// TIA Portal V15.1 export
// export: Created 2020-06-12T07:35:42.9130859Z, ExportSetting None, DisplayName Totally Integrated Automation Portal, DisplayVersion V15.1, DisplayName TIA Portal Openness, DisplayVersion V15.1, DisplayName STEP 7 Professional, DisplayVersion V15.1, DisplayName STEP 7 Safety, DisplayVersion V15.1, DisplayName WinCC Advanced, DisplayVersion V15.1
FUNCTION "CW_MS1" : Void   // FC119, FBD
TITLE = Meltstation #1 cooling control
{ S7_Optimized_Access := 'TRUE' }
// stored: SetENOAutomatically False
   VAR_TEMP
      tContReset : Bool;
      tContDTOn : Bool;
      tMoldIsClosed : Bool;
      tMoldIsOpened : Bool;
      tMoldIsDischarging : Bool;
      tMoldIsPrepared : Bool;
      tBaseIsClosed : Bool;
      tBaseIsOpened : Bool;
      tBaseIsPrepared : Bool;
      tBaseIsDischarging : Bool;
      tLinesToOpen : Bool;
      tLinesToCLose : Bool;
      tToDischarge : Bool;
      tCoolingIsOn : Bool;
      tCoolingOn : Bool;
      tCoolingOff : Bool;
      tCoolingLockOff : Bool;
      tDeltaContOn : Bool;
      tStepError : Bool;
      tReqOn : Bool;
      tReqOff : Bool;
      tReqDisStop : Bool;
      tReqDisStart : Bool;
      tValid : Bool;
      tReqContFlow : Bool;
      tReqContDT : Bool;
      tStage : Int;
      tStepInternal : Int;
      tMoldFlowMax : Real;
      tBaseFlowMax : Real;
      tMoldFlowSet : Real;
      tMoldFlowPhysMax : Real;
      tMoldFlowPhysMin : Real;
      tMoldFlowMin : Real;
      tBaseFlowPhysMax : Real;
      tBaseFlowPhysMin : Real;
      tBaseFlowMin : Real;
      tBaseFlowSet : Real;
      tMoldFlowContIsOn : Bool;
      tBaseFlowContOn : Bool;
      tMoldFlowContIsAuto : Bool;
      tEnAlarms : Bool;
      tCopyParam : Bool;
   END_VAR
BEGIN

REGION Network 1: HMI request treat
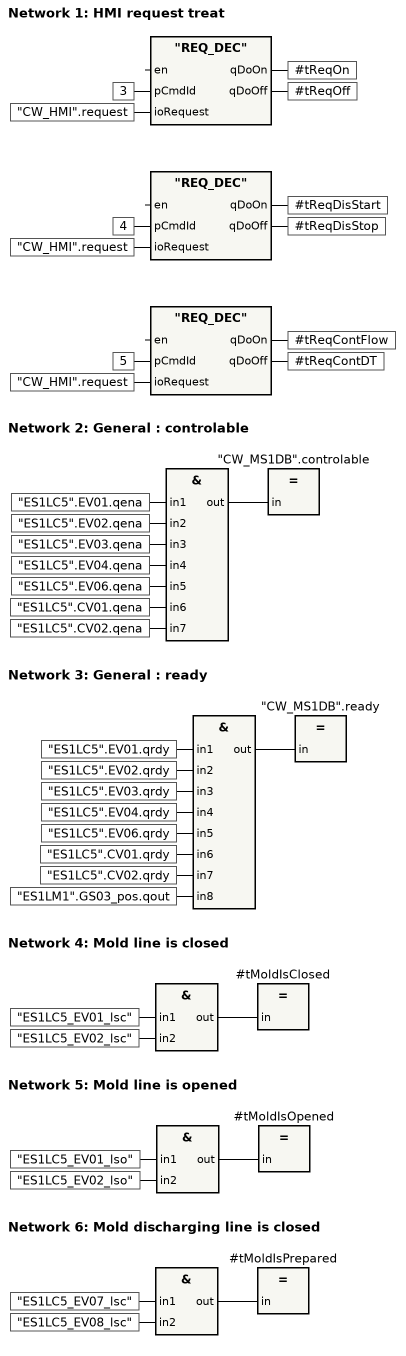
   "REQ_DEC"(pCmdId := 3, ioRequest := "CW_HMI".request, qDoOn => #tReqOn, qDoOff => #tReqOff);
   "REQ_DEC"(pCmdId := 4, ioRequest := "CW_HMI".request, qDoOn => #tReqDisStart, qDoOff => #tReqDisStop);
   "REQ_DEC"(pCmdId := 5, ioRequest := "CW_HMI".request, qDoOn => #tReqContFlow, qDoOff => #tReqContDT);
END_REGION

REGION Network 2: General : controlable
   "CW_MS1DB".controlable := "ES1LC5".EV01.qena AND "ES1LC5".EV02.qena AND "ES1LC5".EV03.qena AND "ES1LC5".EV04.qena AND "ES1LC5".EV06.qena AND "ES1LC5".CV01.qena AND "ES1LC5".CV02.qena;
END_REGION

REGION Network 3: General : ready
   "CW_MS1DB".ready := "ES1LC5".EV01.qrdy AND "ES1LC5".EV02.qrdy AND "ES1LC5".EV03.qrdy AND "ES1LC5".EV04.qrdy AND "ES1LC5".EV06.qrdy AND "ES1LC5".CV01.qrdy AND "ES1LC5".CV02.qrdy AND "ES1LM1".GS03_pos.qout;
END_REGION

REGION Network 4: Mold line is closed
   #tMoldIsClosed := "ES1LC5_EV01_lsc" AND "ES1LC5_EV02_lsc";
END_REGION

REGION Network 5: Mold line is opened
   #tMoldIsOpened := "ES1LC5_EV01_lso" AND "ES1LC5_EV02_lso";
END_REGION

REGION Network 6: Mold discharging line is closed
   #tMoldIsPrepared := "ES1LC5_EV07_lsc" AND "ES1LC5_EV08_lsc";
END_REGION

REGION Network 7: Mold discharging line is opened
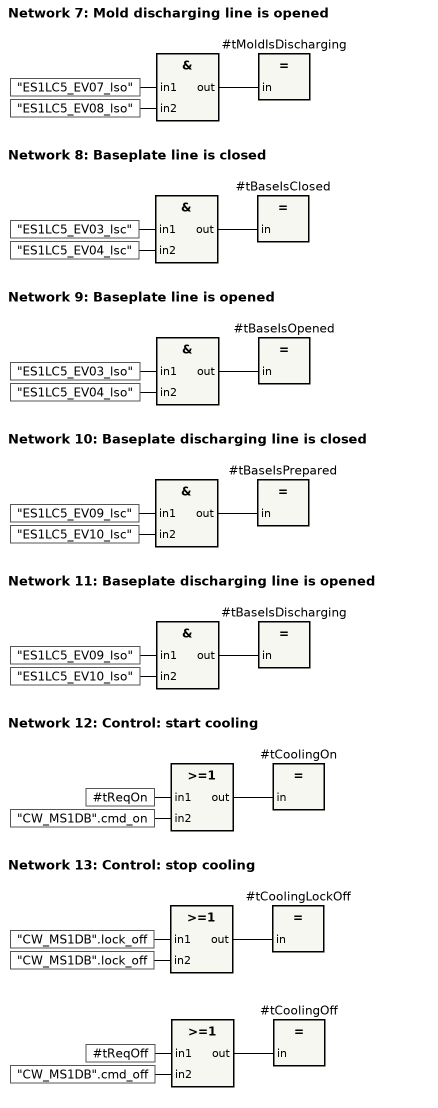
   #tMoldIsDischarging := "ES1LC5_EV07_lso" AND "ES1LC5_EV08_lso";
END_REGION

REGION Network 8: Baseplate line is closed
   #tBaseIsClosed := "ES1LC5_EV03_lsc" AND "ES1LC5_EV04_lsc";
END_REGION

REGION Network 9: Baseplate line is opened
   #tBaseIsOpened := "ES1LC5_EV03_lso" AND "ES1LC5_EV04_lso";
END_REGION

REGION Network 10: Baseplate discharging line is closed
   #tBaseIsPrepared := "ES1LC5_EV09_lsc" AND "ES1LC5_EV10_lsc";
END_REGION

REGION Network 11: Baseplate discharging line is opened
   #tBaseIsDischarging := "ES1LC5_EV09_lso" AND "ES1LC5_EV10_lso";
END_REGION

REGION Network 12: Control: start cooling
   #tCoolingOn := #tReqOn OR "CW_MS1DB".cmd_on;
END_REGION

REGION Network 13: Control: stop cooling
   // #tReqAmcOff
   #tCoolingLockOff := "CW_MS1DB".lock_off OR "CW_MS1DB".lock_off;
   #tCoolingOff := #tReqOff OR "CW_MS1DB".cmd_off;
END_REGION

REGION Network 14: *** Control (stages) ***
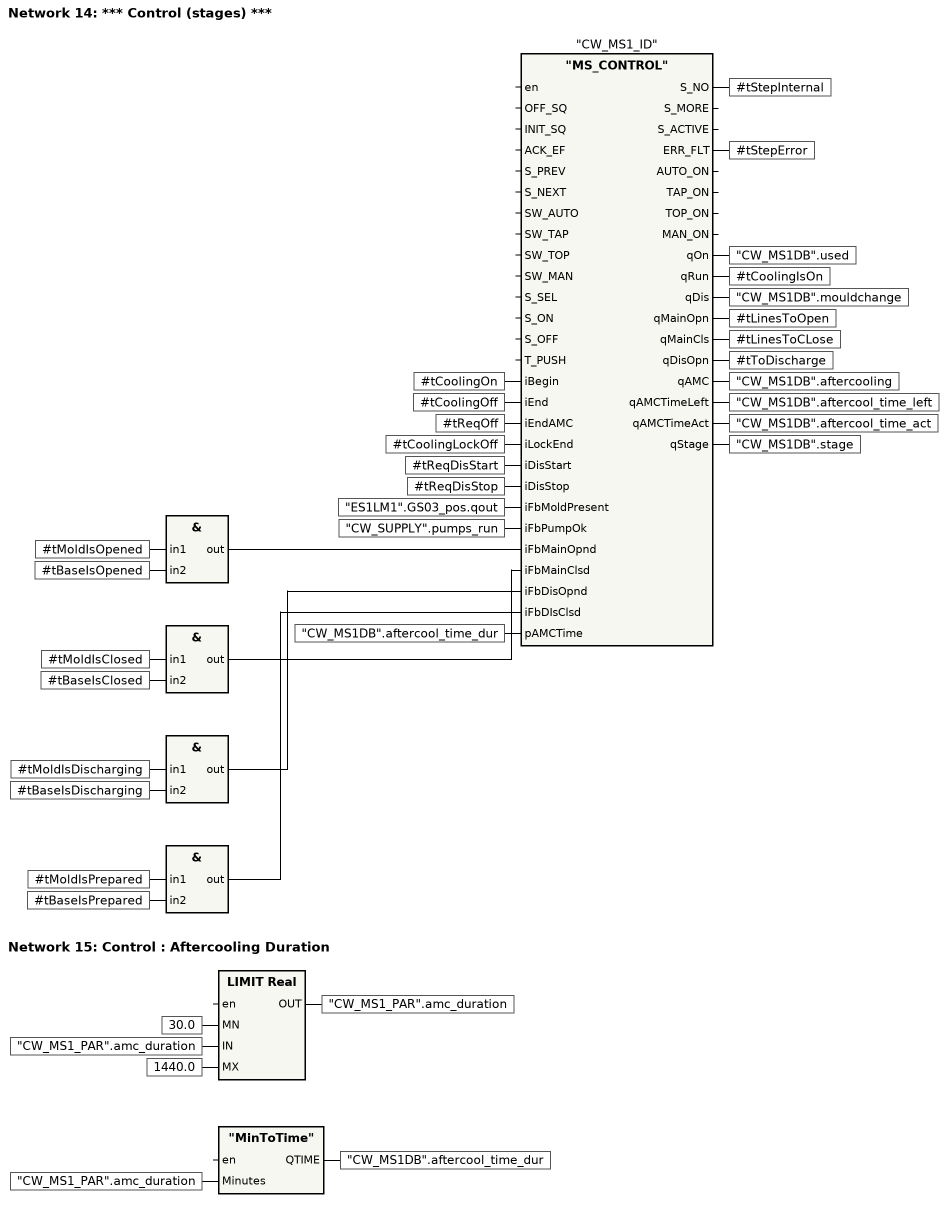
   "CW_MS1_ID"(iBegin := #tCoolingOn,   // "MS_CONTROL"
               iEnd := #tCoolingOff,
               iEndAMC := #tReqOff,
               iLockEnd := #tCoolingLockOff,
               iDisStart := #tReqDisStart,
               iDisStop := #tReqDisStop,
               iFbMoldPresent := "ES1LM1".GS03_pos.qout,
               iFbPumpOk := "CW_SUPPLY".pumps_run,
               iFbMainOpnd := #tMoldIsOpened AND #tBaseIsOpened,
               iFbMainClsd := #tMoldIsClosed AND #tBaseIsClosed,
               iFbDisOpnd := #tMoldIsDischarging AND #tBaseIsDischarging,
               iFbDIsClsd := #tMoldIsPrepared AND #tBaseIsPrepared,
               pAMCTime := "CW_MS1DB".aftercool_time_dur,
               S_NO => #tStepInternal,
               ERR_FLT => #tStepError,
               qOn => "CW_MS1DB".used,
               qRun => #tCoolingIsOn,
               qDis => "CW_MS1DB".mouldchange,
               qMainOpn => #tLinesToOpen,
               qMainCls => #tLinesToCLose,
               qDisOpn => #tToDischarge,
               qAMC => "CW_MS1DB".aftercooling,
               qAMCTimeLeft => "CW_MS1DB".aftercool_time_left,
               qAMCTimeAct => "CW_MS1DB".aftercool_time_act,
               qStage => "CW_MS1DB".stage);
END_REGION

REGION Network 15: Control : Aftercooling Duration
   // Convert minutes to milliseconds
   "CW_MS1_PAR".amc_duration := LIMIT(MN := 30.0, IN := "CW_MS1_PAR".amc_duration, MX := 1440.0);
   "MinToTime"(Minutes := "CW_MS1_PAR".amc_duration, QTIME => "CW_MS1DB".aftercool_time_dur);
END_REGION

REGION Network 16: Cooling mode: flow/delta-T
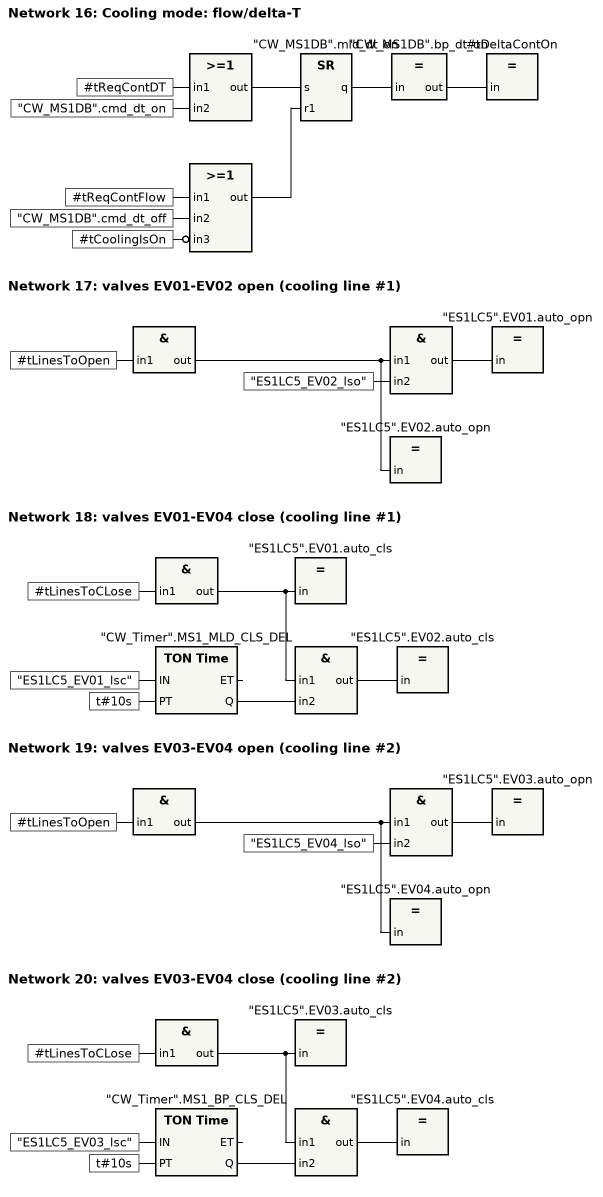
   IF #tReqContDT OR "CW_MS1DB".cmd_dt_on THEN
       "CW_MS1DB".mld_dt_on := TRUE;   // SR flip-flop
   END_IF;
   IF #tReqContFlow OR "CW_MS1DB".cmd_dt_off OR NOT #tCoolingIsOn THEN "CW_MS1DB".mld_dt_on := FALSE; END_IF;
   "CW_MS1DB".bp_dt_on := "CW_MS1DB".mld_dt_on;
   #tDeltaContOn := "CW_MS1DB".mld_dt_on;
END_REGION

REGION Network 17: valves EV01-EV02 open (cooling line #1)
   "ES1LC5".EV01.auto_opn := #tLinesToOpen AND "ES1LC5_EV02_lso";
   "ES1LC5".EV02.auto_opn := #tLinesToOpen;
END_REGION

REGION Network 18: valves EV01-EV04 close (cooling line #1)
   "ES1LC5".EV01.auto_cls := #tLinesToCLose;
   "CW_Timer".MS1_MLD_CLS_DEL.TON(IN := "ES1LC5_EV01_lsc", PT := t#10s);
   "ES1LC5".EV02.auto_cls := #tLinesToCLose AND "CW_Timer".MS1_MLD_CLS_DEL.Q;
END_REGION

REGION Network 19: valves EV03-EV04 open (cooling line #2)
   "ES1LC5".EV03.auto_opn := #tLinesToOpen AND "ES1LC5_EV04_lso";
   "ES1LC5".EV04.auto_opn := #tLinesToOpen;
END_REGION

REGION Network 20: valves EV03-EV04 close (cooling line #2)
   "ES1LC5".EV03.auto_cls := #tLinesToCLose;
   "CW_Timer".MS1_BP_CLS_DEL.TON(IN := "ES1LC5_EV03_lsc", PT := t#10s);
   "ES1LC5".EV04.auto_cls := #tLinesToCLose AND "CW_Timer".MS1_BP_CLS_DEL.Q;
END_REGION

REGION Network 21: valves EV01-EV04 to close lock
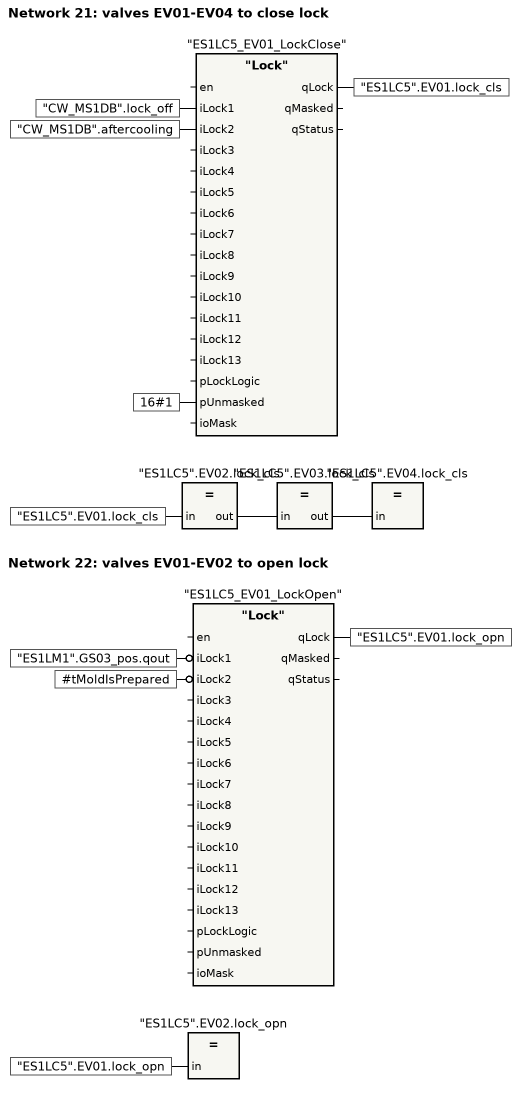
   "ES1LC5_EV01_LockClose"(iLock1 := "CW_MS1DB".lock_off,   // "Lock"
                           iLock2 := "CW_MS1DB".aftercooling,
                           pUnmasked := 16#1,
                           qLock => "ES1LC5".EV01.lock_cls);
   "ES1LC5".EV02.lock_cls := "ES1LC5".EV01.lock_cls;
   "ES1LC5".EV03.lock_cls := "ES1LC5".EV01.lock_cls;
   "ES1LC5".EV04.lock_cls := "ES1LC5".EV01.lock_cls;
END_REGION

REGION Network 22: valves EV01-EV02 to open lock
   "ES1LC5_EV01_LockOpen"(iLock1 := NOT "ES1LM1".GS03_pos.qout,   // "Lock"
                          iLock2 := NOT #tMoldIsPrepared,
                          qLock => "ES1LC5".EV01.lock_opn);
   "ES1LC5".EV02.lock_opn := "ES1LC5".EV01.lock_opn;
END_REGION

REGION Network 23: valves EV03-EV04 to open lock
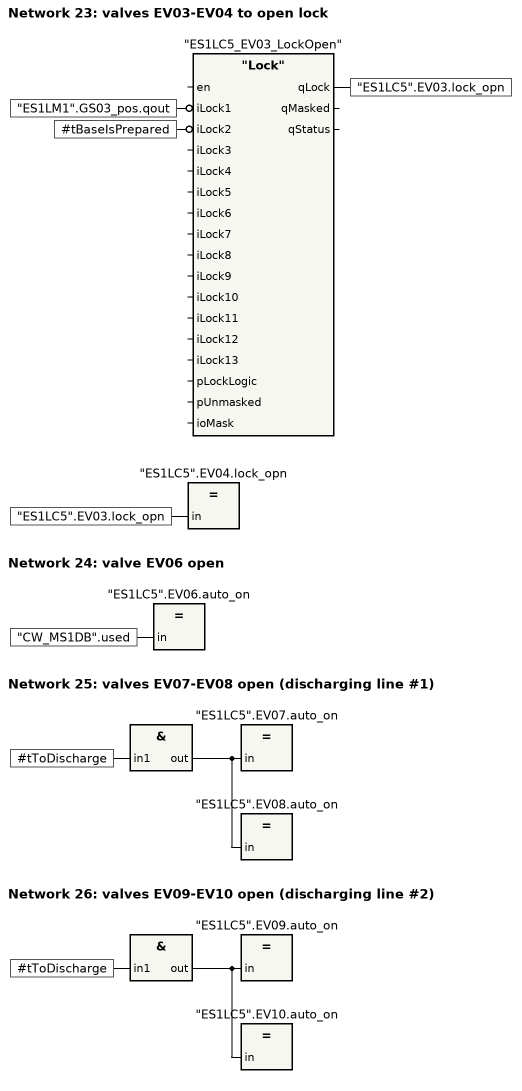
   "ES1LC5_EV03_LockOpen"(iLock1 := NOT "ES1LM1".GS03_pos.qout,   // "Lock"
                          iLock2 := NOT #tBaseIsPrepared,
                          qLock => "ES1LC5".EV03.lock_opn);
   "ES1LC5".EV04.lock_opn := "ES1LC5".EV03.lock_opn;
END_REGION

REGION Network 24: valve EV06 open
   "ES1LC5".EV06.auto_on := "CW_MS1DB".used;
END_REGION

REGION Network 25: valves EV07-EV08 open (discharging line #1)
   "ES1LC5".EV07.auto_on := #tToDischarge;
   "ES1LC5".EV08.auto_on := #tToDischarge;
END_REGION

REGION Network 26: valves EV09-EV10 open (discharging line #2)
   "ES1LC5".EV09.auto_on := #tToDischarge;
   "ES1LC5".EV10.auto_on := #tToDischarge;
END_REGION

REGION Network 27: valves EV07-EV08 to open lock (discharging line #1)
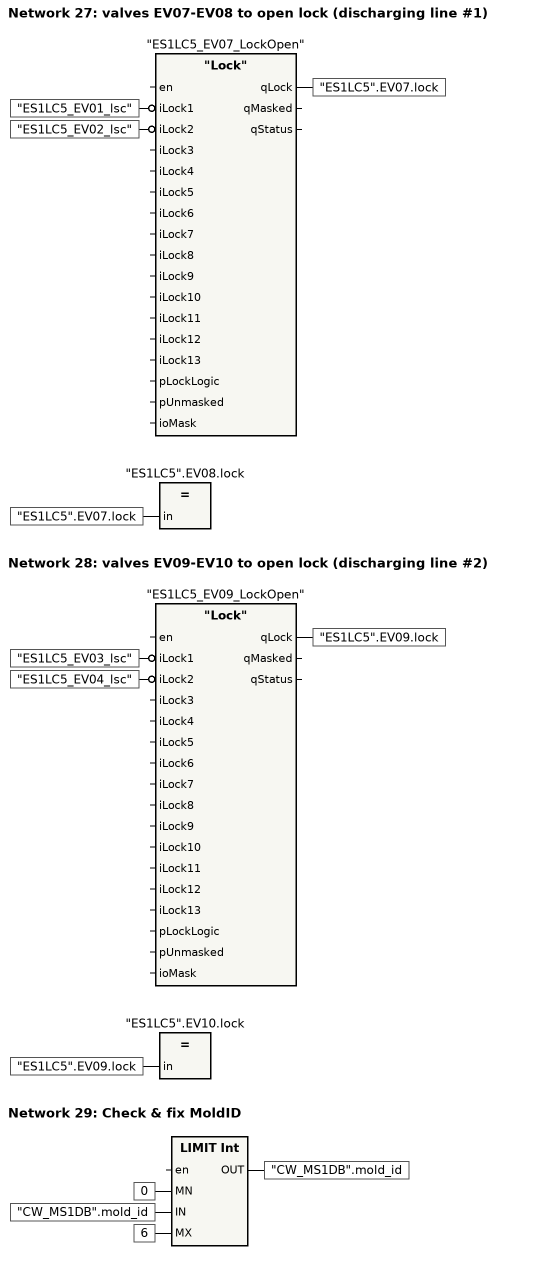
   "ES1LC5_EV07_LockOpen"(iLock1 := NOT "ES1LC5_EV01_lsc",   // "Lock"
                          iLock2 := NOT "ES1LC5_EV02_lsc",
                          qLock => "ES1LC5".EV07.lock);
   "ES1LC5".EV08.lock := "ES1LC5".EV07.lock;
END_REGION

REGION Network 28: valves EV09-EV10 to open lock (discharging line #2)
   "ES1LC5_EV09_LockOpen"(iLock1 := NOT "ES1LC5_EV03_lsc",   // "Lock"
                          iLock2 := NOT "ES1LC5_EV04_lsc",
                          qLock => "ES1LC5".EV09.lock);
   "ES1LC5".EV10.lock := "ES1LC5".EV09.lock;
END_REGION

REGION Network 29: Check & fix MoldID
   "CW_MS1DB".mold_id := LIMIT(MN := 0, IN := "CW_MS1DB".mold_id, MX := 6);
END_REGION

REGION Network 30: MOULD: Setpoint flow mould
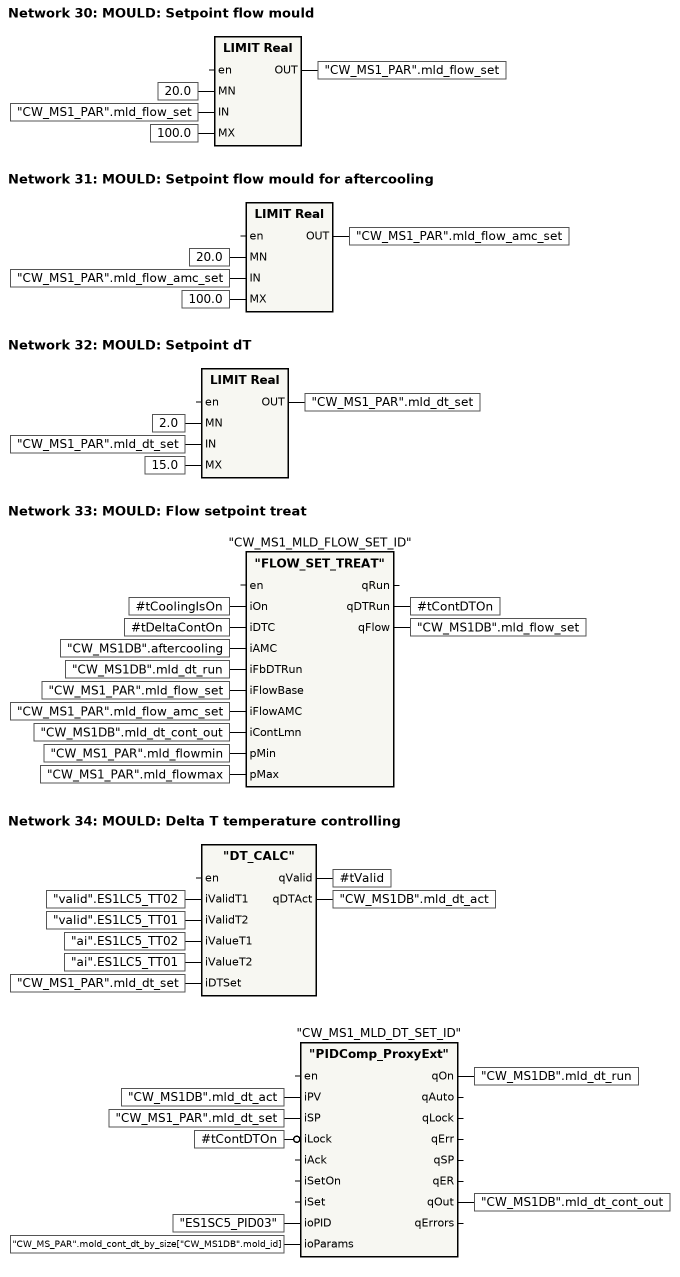
   "CW_MS1_PAR".mld_flow_set := LIMIT(MN := 20.0, IN := "CW_MS1_PAR".mld_flow_set, MX := 100.0);
END_REGION

REGION Network 31: MOULD: Setpoint flow mould for aftercooling
   "CW_MS1_PAR".mld_flow_amc_set := LIMIT(MN := 20.0, IN := "CW_MS1_PAR".mld_flow_amc_set, MX := 100.0);
END_REGION

REGION Network 32: MOULD: Setpoint dT
   "CW_MS1_PAR".mld_dt_set := LIMIT(MN := 2.0, IN := "CW_MS1_PAR".mld_dt_set, MX := 15.0);
END_REGION

REGION Network 33: MOULD: Flow setpoint treat
   "CW_MS1_MLD_FLOW_SET_ID"(iOn := #tCoolingIsOn,   // "FLOW_SET_TREAT"
                           iDTC := #tDeltaContOn,
                           iAMC := "CW_MS1DB".aftercooling,
                           iFbDTRun := "CW_MS1DB".mld_dt_run,
                           iFlowBase := "CW_MS1_PAR".mld_flow_set,
                           iFlowAMC := "CW_MS1_PAR".mld_flow_amc_set,
                           iContLmn := "CW_MS1DB".mld_dt_cont_out,
                           pMin := "CW_MS1_PAR".mld_flowmin,
                           pMax := "CW_MS1_PAR".mld_flowmax,
                           qDTRun => #tContDTOn,
                           qFlow => "CW_MS1DB".mld_flow_set);
END_REGION

REGION Network 34: MOULD: Delta T temperature controlling
   "DT_CALC"(iValidT1 := "valid".ES1LC5_TT02,
             iValidT2 := "valid".ES1LC5_TT01,
             iValueT1 := "ai".ES1LC5_TT02,
             iValueT2 := "ai".ES1LC5_TT01,
             iDTSet := "CW_MS1_PAR".mld_dt_set,
             qValid => #tValid,
             qDTAct => "CW_MS1DB".mld_dt_act);
   "CW_MS1_MLD_DT_SET_ID"(iPV := "CW_MS1DB".mld_dt_act,   // "PIDComp_ProxyExt"
                          iSP := "CW_MS1_PAR".mld_dt_set,
                          iLock := NOT #tContDTOn,
                          ioPID := "ES1SC5_PID03",
                          ioParams := "CW_MS_PAR".mold_cont_dt_by_size["CW_MS1DB".mold_id],
                          qOn => "CW_MS1DB".mld_dt_run,
                          qOut => "CW_MS1DB".mld_dt_cont_out);
END_REGION

REGION Network 35: MOULD: Flow Controller
   // Yes, the actual value is keeping while a measurement is not valid.
   // If the controller is stable (ERR = 0) we can avoid a bump by flow,
   // else if ERR > 0 the controller will open the valve, and this is also not bad
   // else the controller will close the valve, and this is bad...
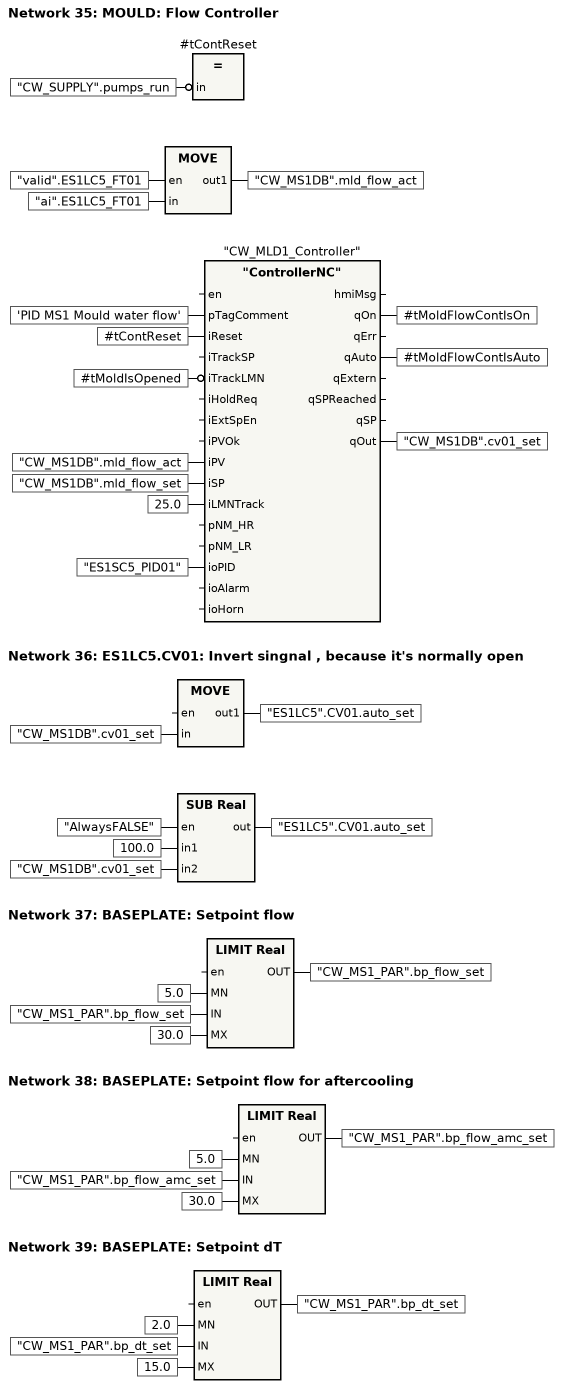
   #tContReset := NOT "CW_SUPPLY".pumps_run;
   IF "valid".ES1LC5_FT01 THEN "CW_MS1DB".mld_flow_act := "ai".ES1LC5_FT01; END_IF;
   "CW_MLD1_Controller"(pTagComment := 'PID MS1 Mould water flow',   // "ControllerNC"
                        iReset := #tContReset,
                        iTrackLMN := NOT #tMoldIsOpened,
                        iPV := "CW_MS1DB".mld_flow_act,
                        iSP := "CW_MS1DB".mld_flow_set,
                        iLMNTrack := 25.0,
                        ioPID := "ES1SC5_PID01",
                        qOn => #tMoldFlowContIsOn,
                        qAuto => #tMoldFlowContIsAuto,
                        qOut => "CW_MS1DB".cv01_set);
END_REGION

REGION Network 36: ES1LC5.CV01: Invert singnal , because it's normally open
   "ES1LC5".CV01.auto_set := "CW_MS1DB".cv01_set;
   IF "AlwaysFALSE" THEN "ES1LC5".CV01.auto_set := 100.0 - "CW_MS1DB".cv01_set; END_IF;
END_REGION

REGION Network 37: BASEPLATE: Setpoint flow
   "CW_MS1_PAR".bp_flow_set := LIMIT(MN := 5.0, IN := "CW_MS1_PAR".bp_flow_set, MX := 30.0);
END_REGION

REGION Network 38: BASEPLATE: Setpoint flow for aftercooling
   "CW_MS1_PAR".bp_flow_amc_set := LIMIT(MN := 5.0, IN := "CW_MS1_PAR".bp_flow_amc_set, MX := 30.0);
END_REGION

REGION Network 39: BASEPLATE: Setpoint dT
   "CW_MS1_PAR".bp_dt_set := LIMIT(MN := 2.0, IN := "CW_MS1_PAR".bp_dt_set, MX := 15.0);
END_REGION

REGION Network 40: BASEPLATE: Flow setpoint treat
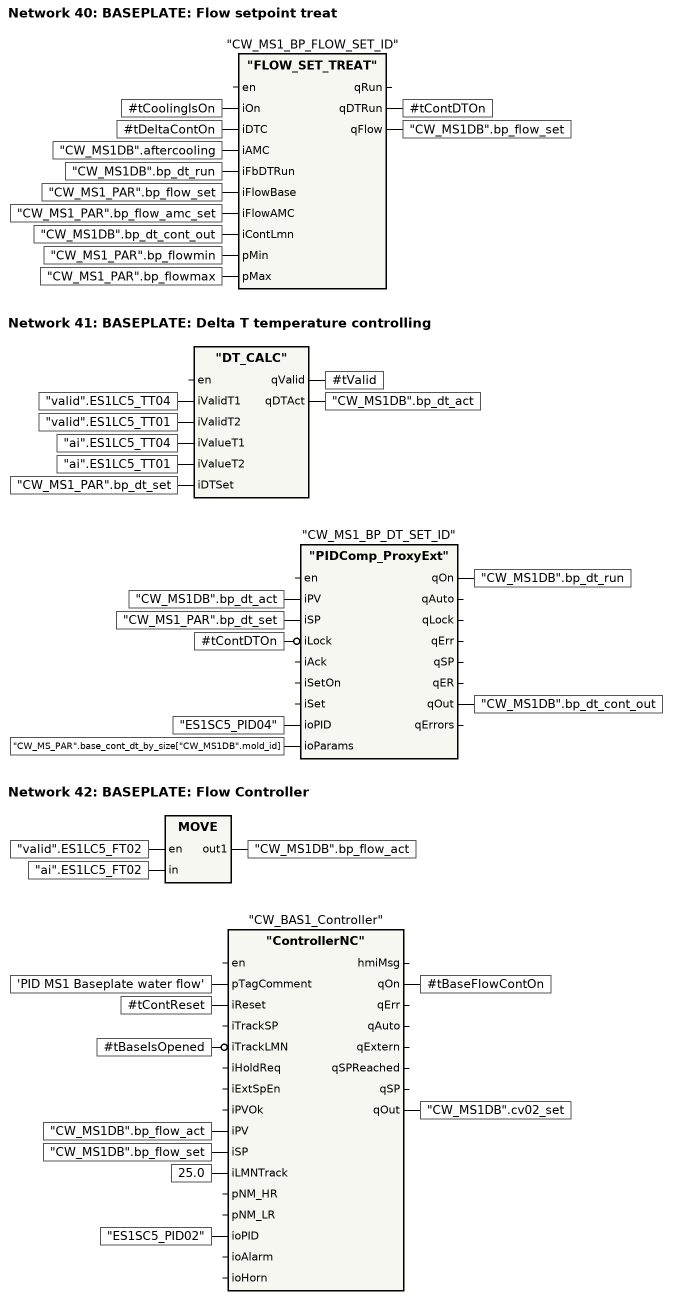
   "CW_MS1_BP_FLOW_SET_ID"(iOn := #tCoolingIsOn,   // "FLOW_SET_TREAT"
                           iDTC := #tDeltaContOn,
                           iAMC := "CW_MS1DB".aftercooling,
                           iFbDTRun := "CW_MS1DB".bp_dt_run,
                           iFlowBase := "CW_MS1_PAR".bp_flow_set,
                           iFlowAMC := "CW_MS1_PAR".bp_flow_amc_set,
                           iContLmn := "CW_MS1DB".bp_dt_cont_out,
                           pMin := "CW_MS1_PAR".bp_flowmin,
                           pMax := "CW_MS1_PAR".bp_flowmax,
                           qDTRun => #tContDTOn,
                           qFlow => "CW_MS1DB".bp_flow_set);
END_REGION

REGION Network 41: BASEPLATE: Delta T temperature controlling
   // TODO Adapter-Function for selecting PID-parameters with TUNING-option
   "DT_CALC"(iValidT1 := "valid".ES1LC5_TT04,
             iValidT2 := "valid".ES1LC5_TT01,
             iValueT1 := "ai".ES1LC5_TT04,
             iValueT2 := "ai".ES1LC5_TT01,
             iDTSet := "CW_MS1_PAR".bp_dt_set,
             qValid => #tValid,
             qDTAct => "CW_MS1DB".bp_dt_act);
   "CW_MS1_BP_DT_SET_ID"(iPV := "CW_MS1DB".bp_dt_act,   // "PIDComp_ProxyExt"
                         iSP := "CW_MS1_PAR".bp_dt_set,
                         iLock := NOT #tContDTOn,
                         ioPID := "ES1SC5_PID04",
                         ioParams := "CW_MS_PAR".base_cont_dt_by_size["CW_MS1DB".mold_id],
                         qOn => "CW_MS1DB".bp_dt_run,
                         qOut => "CW_MS1DB".bp_dt_cont_out);
END_REGION

REGION Network 42: BASEPLATE: Flow Controller
   // Yes, the actual value is keeping while a measurement is not valid.
   // If the controller is stable (ERR = 0) we can avoid a bump by flow,
   // else if ERR > 0 the controller will open the valve, and this is also not bad
   // else the controller will close the valve, and this is bad...
   IF "valid".ES1LC5_FT02 THEN "CW_MS1DB".bp_flow_act := "ai".ES1LC5_FT02; END_IF;
   "CW_BAS1_Controller"(pTagComment := 'PID MS1 Baseplate water flow',   // "ControllerNC"
                        iReset := #tContReset,
                        iTrackLMN := NOT #tBaseIsOpened,
                        iPV := "CW_MS1DB".bp_flow_act,
                        iSP := "CW_MS1DB".bp_flow_set,
                        iLMNTrack := 25.0,
                        ioPID := "ES1SC5_PID02",
                        qOn => #tBaseFlowContOn,
                        qOut => "CW_MS1DB".cv02_set);
END_REGION

REGION Network 43: ES1LC5.CV02: Invert singnal , because it's normally open
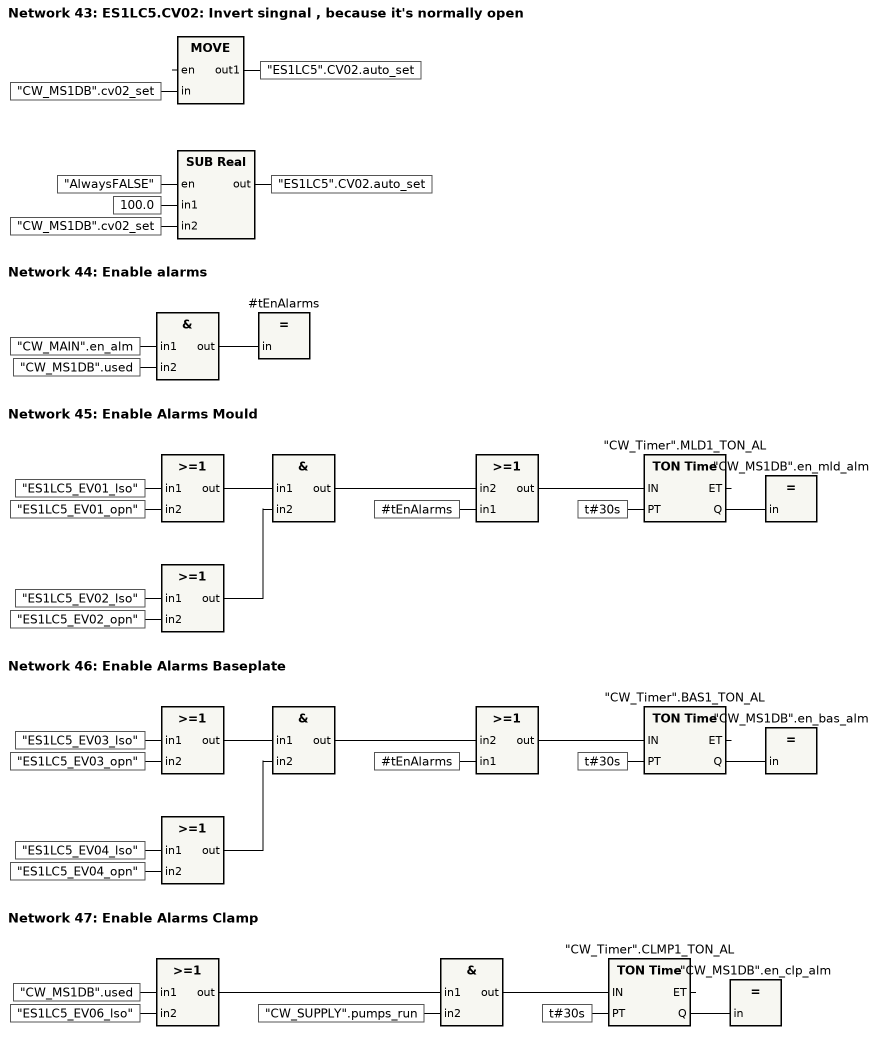
   "ES1LC5".CV02.auto_set := "CW_MS1DB".cv02_set;
   IF "AlwaysFALSE" THEN "ES1LC5".CV02.auto_set := 100.0 - "CW_MS1DB".cv02_set; END_IF;
END_REGION

REGION Network 44: Enable alarms
   #tEnAlarms := "CW_MAIN".en_alm AND "CW_MS1DB".used;
END_REGION

REGION Network 45: Enable Alarms Mould
   "CW_Timer".MLD1_TON_AL.TON(IN := (("ES1LC5_EV01_lso" OR "ES1LC5_EV01_opn") AND ("ES1LC5_EV02_lso" OR "ES1LC5_EV02_opn")) OR #tEnAlarms,
                           PT := t#30s);
   "CW_MS1DB".en_mld_alm := "CW_Timer".MLD1_TON_AL.Q;
END_REGION

REGION Network 46: Enable Alarms Baseplate
   "CW_Timer".BAS1_TON_AL.TON(IN := (("ES1LC5_EV03_lso" OR "ES1LC5_EV03_opn") AND ("ES1LC5_EV04_lso" OR "ES1LC5_EV04_opn")) OR #tEnAlarms,
                           PT := t#30s);
   "CW_MS1DB".en_bas_alm := "CW_Timer".BAS1_TON_AL.Q;
END_REGION

REGION Network 47: Enable Alarms Clamp
   "CW_Timer".CLMP1_TON_AL.TON(IN := ("CW_MS1DB".used OR "ES1LC5_EV06_lso") AND "CW_SUPPLY".pumps_run,
                           PT := t#30s);
   "CW_MS1DB".en_clp_alm := "CW_Timer".CLMP1_TON_AL.Q;
END_REGION

REGION Network 48: HMI: STATUS
   // #tMoldFlowContIsOn
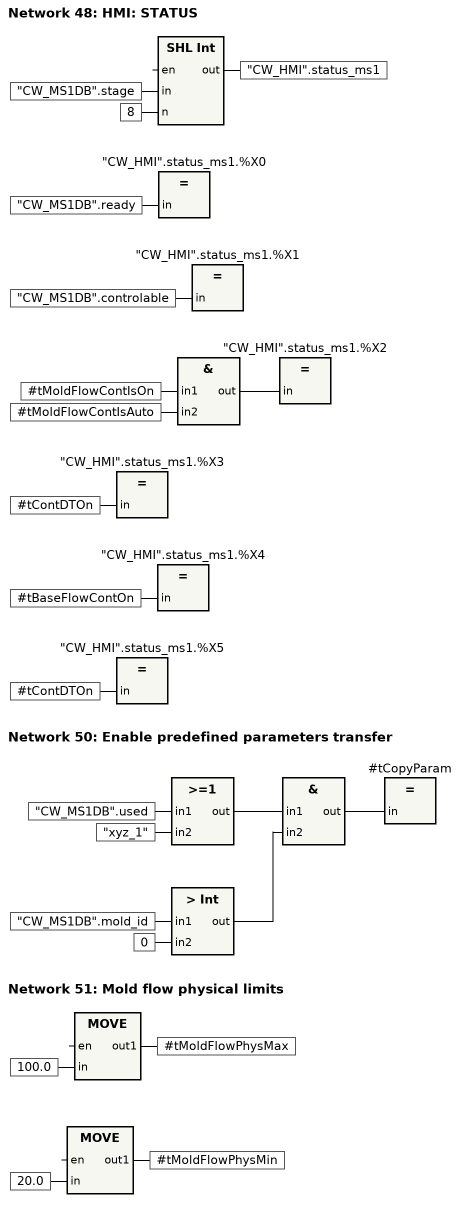
   "CW_HMI".status_ms1 := SHL(IN := "CW_MS1DB".stage, N := 8);
   "CW_HMI".status_ms1.%X0 := "CW_MS1DB".ready;
   "CW_HMI".status_ms1.%X1 := "CW_MS1DB".controlable;
   "CW_HMI".status_ms1.%X2 := #tMoldFlowContIsOn AND #tMoldFlowContIsAuto;
   "CW_HMI".status_ms1.%X3 := #tContDTOn;
   "CW_HMI".status_ms1.%X4 := #tBaseFlowContOn;
   "CW_HMI".status_ms1.%X5 := #tContDTOn;
END_REGION

REGION Network 49: [PAPARMETERS selection]
END_REGION

REGION Network 50: Enable predefined parameters transfer
   #tCopyParam := ("CW_MS1DB".used OR "xyz_1") AND ("CW_MS1DB".mold_id > 0);
END_REGION

REGION Network 51: Mold flow physical limits
   #tMoldFlowPhysMax := 100.0;
   #tMoldFlowPhysMin := 20.0;
END_REGION

REGION Network 52: Mold max flow limit
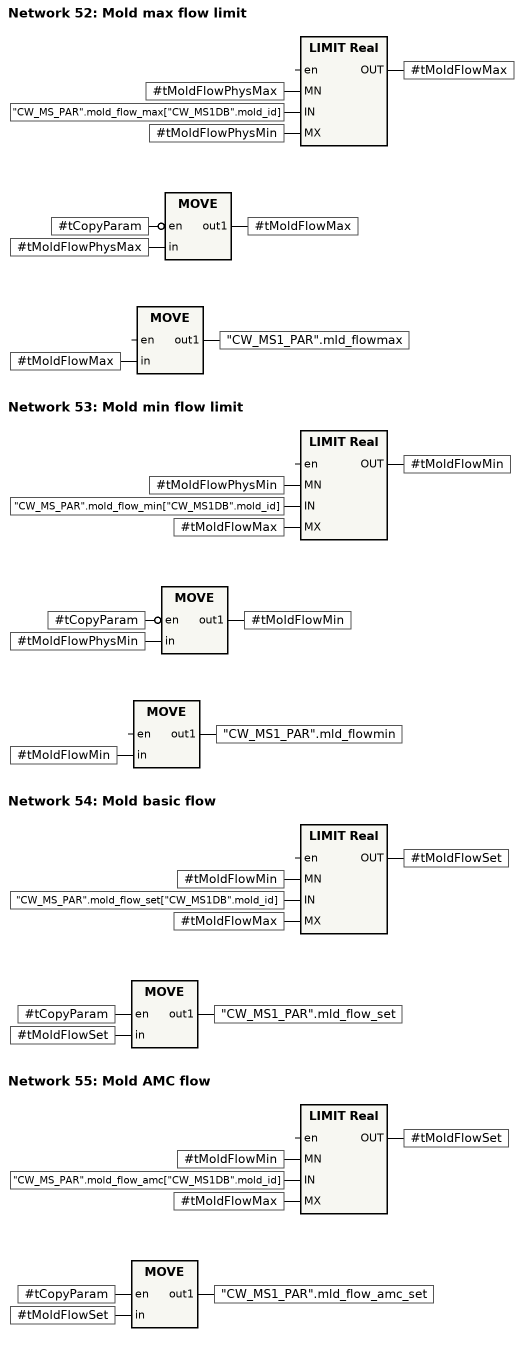
   #tMoldFlowMax := LIMIT(MN := #tMoldFlowPhysMax, IN := "CW_MS_PAR".mold_flow_max["CW_MS1DB".mold_id], MX := #tMoldFlowPhysMin);
   IF NOT #tCopyParam THEN #tMoldFlowMax := #tMoldFlowPhysMax; END_IF;
   "CW_MS1_PAR".mld_flowmax := #tMoldFlowMax;
END_REGION

REGION Network 53: Mold min flow limit
   #tMoldFlowMin := LIMIT(MN := #tMoldFlowPhysMin, IN := "CW_MS_PAR".mold_flow_min["CW_MS1DB".mold_id], MX := #tMoldFlowMax);
   IF NOT #tCopyParam THEN #tMoldFlowMin := #tMoldFlowPhysMin; END_IF;
   "CW_MS1_PAR".mld_flowmin := #tMoldFlowMin;
END_REGION

REGION Network 54: Mold basic flow
   #tMoldFlowSet := LIMIT(MN := #tMoldFlowMin, IN := "CW_MS_PAR".mold_flow_set["CW_MS1DB".mold_id], MX := #tMoldFlowMax);
   IF #tCopyParam THEN "CW_MS1_PAR".mld_flow_set := #tMoldFlowSet; END_IF;
END_REGION

REGION Network 55: Mold AMC flow
   #tMoldFlowSet := LIMIT(MN := #tMoldFlowMin, IN := "CW_MS_PAR".mold_flow_amc["CW_MS1DB".mold_id], MX := #tMoldFlowMax);
   IF #tCopyParam THEN "CW_MS1_PAR".mld_flow_amc_set := #tMoldFlowSet; END_IF;
END_REGION

REGION Network 56: Baseplate flow physical limits
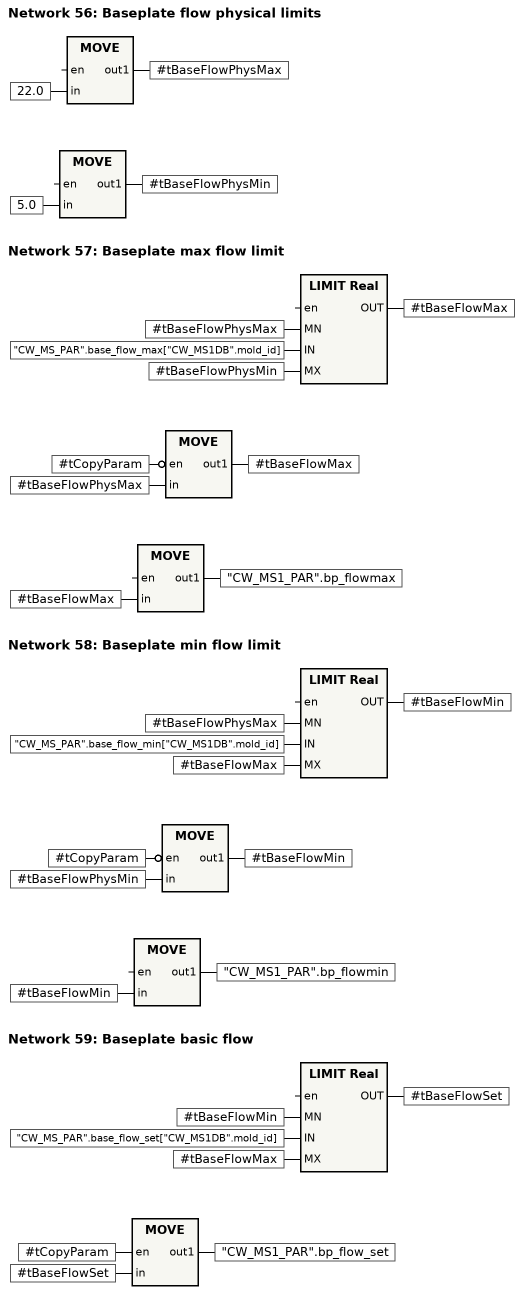
   #tBaseFlowPhysMax := 22.0;
   #tBaseFlowPhysMin := 5.0;
END_REGION

REGION Network 57: Baseplate max flow limit
   #tBaseFlowMax := LIMIT(MN := #tBaseFlowPhysMax, IN := "CW_MS_PAR".base_flow_max["CW_MS1DB".mold_id], MX := #tBaseFlowPhysMin);
   IF NOT #tCopyParam THEN #tBaseFlowMax := #tBaseFlowPhysMax; END_IF;
   "CW_MS1_PAR".bp_flowmax := #tBaseFlowMax;
END_REGION

REGION Network 58: Baseplate min flow limit
   #tBaseFlowMin := LIMIT(MN := #tBaseFlowPhysMax, IN := "CW_MS_PAR".base_flow_min["CW_MS1DB".mold_id], MX := #tBaseFlowMax);
   IF NOT #tCopyParam THEN #tBaseFlowMin := #tBaseFlowPhysMin; END_IF;
   "CW_MS1_PAR".bp_flowmin := #tBaseFlowMin;
END_REGION

REGION Network 59: Baseplate basic flow
   // May be a table using for the setpoint selection is not good idea
   #tBaseFlowSet := LIMIT(MN := #tBaseFlowMin, IN := "CW_MS_PAR".base_flow_set["CW_MS1DB".mold_id], MX := #tBaseFlowMax);
   IF #tCopyParam THEN "CW_MS1_PAR".bp_flow_set := #tBaseFlowSet; END_IF;
END_REGION

REGION Network 60: Baseplate AMC flow
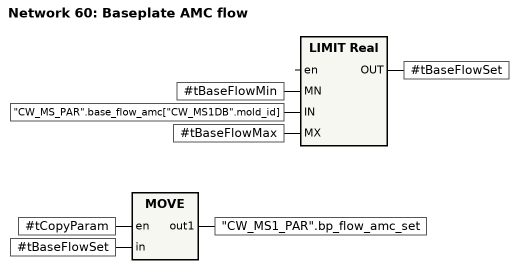
   #tBaseFlowSet := LIMIT(MN := #tBaseFlowMin, IN := "CW_MS_PAR".base_flow_amc["CW_MS1DB".mold_id], MX := #tBaseFlowMax);
   IF #tCopyParam THEN "CW_MS1_PAR".bp_flow_amc_set := #tBaseFlowSet; END_IF;
END_REGION
END_FUNCTION
